DATA_BLOCK "DB_MC2"
{ S7_Optimized_Access := 'TRUE' }
VERSION : 0.1
NON_RETAIN
"FB_MC_Dummy"

BEGIN

END_DATA_BLOCK

